(* IEC 61131-3 sources: volt/packages/volt-lsp-iec/test-corpus/lenze-mid/Device/Plc Logic/Application/Library Manager/(unresolved)/iecvaraccessopcuametadata interfaces, 4 files *)

(* ---- VARACCUANAMESPACEFRAGMENT.dut ---- *)
TYPE VARACCUANAMESPACEFRAGMENT :
STRUCT
	FRAGMENTNAMESPACE : POINTER TO OpcUa_String;
	NAMESPACES : POINTER TO OpcUa_String;
	NUMNAMESPACES : UDINT;
	NODES : POINTER TO OpcUaServerNodeDescription;
	NUMNODES : UDINT;
	REFERENCES : POINTER TO OpcUaServerReferenceDescription;
	NUMREFERENCES : UDINT;
	NAMESPACESMAPPED : BOOL;
	INVALIDFRAGMENT : BOOL;
	REFCOUNT : UDINT;
END_STRUCT
END_TYPE

(* ---- INTERFACEIDS.gvl ---- *)
VAR_GLOBAL
	ITFID_IIECVARACCESSOPCUAMETADATA : DWORD := 16#C0;
	ITFID_IIECVARACCESSOPCUAFINDBYBROWSENAME : DWORD := 16#D1;
END_VAR

(* ---- IIECVARACCESSOPCUAFINDBYBROWSENAME.itf ---- *)
INTERFACE IIECVARACCESSOPCUAFINDBYBROWSENAME
END_INTERFACE

METHOD VARACCGETCHILDBYBROWSENAME : IBaseTreeNode
VAR_INPUT
	HNODE : RTS_IEC_HANDLE;
	PVARIABLEINFORMATION : POINTER TO VariableInformationStruct2;
	PBROWSENAME : POINTER TO OpcUa_QualifiedName;
	PRESULT : POINTER TO UDINT;
END_VAR
END_METHOD

METHOD VARACCGETNEXTBYBROWSENAME : IBaseTreeNode
VAR_INPUT
	HNODE : RTS_IEC_HANDLE;
	PVARIABLEINFORMATION : POINTER TO VariableInformationStruct2;
	PBROWSENAME : POINTER TO OpcUa_QualifiedName;
	PRESULT : POINTER TO UDINT;
END_VAR
END_METHOD

(* ---- IIECVARACCESSOPCUAMETADATA.itf ---- *)
INTERFACE IIECVARACCESSOPCUAMETADATA
END_INTERFACE

METHOD VARACCGETUAINFORMATIONMODEL : RTS_IEC_RESULT
VAR_OUTPUT
	NAMESPACES : POINTER TO OpcUa_String;
	NUMNAMESPACES : UDINT;
	FRAGMENTS : POINTER TO POINTER TO VarAccUaNamespaceFragment;
	NUMFRAGMENTS : UDINT;
END_VAR
END_METHOD

METHOD VARACCGETUANAMESPACE : RTS_IEC_RESULT
VAR_OUTPUT
	PMODELNAMESPACE : POINTER TO OpcUa_String;
END_VAR
END_METHOD

METHOD VARACCGETUAENTRYPOINTS : RTS_IEC_RESULT
VAR_OUTPUT
	ENTRYPOINTS : POINTER TO OpcUa_NodeId;
	NUMENTRYPOINTS : UDINT;
END_VAR
END_METHOD

METHOD VARACCGETUAMETHODARGUMENTS : RTS_IEC_RESULT
VAR_INPUT
	HNODE : RTS_IEC_HANDLE;
	PVARINFO : POINTER TO VariableInformationStruct2;
END_VAR
VAR_OUTPUT
	PINPUTARGUMENTS : POINTER TO OpcUa_NodeId;
	POUTPUTARGUMENTS : POINTER TO OpcUa_NodeId;
END_VAR
END_METHOD

METHOD VARACCGETUAENTRYPOINT : RTS_IEC_RESULT
VAR_INPUT
	HNODE : RTS_IEC_HANDLE;
	PVARINFO : POINTER TO VariableInformationStruct2;
END_VAR
VAR_OUTPUT
	ISENTRYPOINT : BOOL;
	PENTRYPOINT : POINTER TO OpcUa_NodeId;
END_VAR
END_METHOD

METHOD VARACCGETUAPARENTREFERENCETYPE : RTS_IEC_RESULT
VAR_INPUT
	HNODE : RTS_IEC_HANDLE;
	PVARINFO : POINTER TO VariableInformationStruct2;
END_VAR
VAR_OUTPUT
	PREFERENCETYPE : POINTER TO OpcUa_NodeId;
END_VAR
END_METHOD

METHOD VARACCGETUATYPEDEFINITION : RTS_IEC_RESULT
VAR_INPUT
	HNODE : RTS_IEC_HANDLE;
	PVARINFO : POINTER TO VariableInformationStruct2;
END_VAR
VAR_OUTPUT
	PTYPEDEFINITION : POINTER TO OpcUa_NodeId;
END_VAR
END_METHOD

METHOD VARACCGETUANODECLASS : RTS_IEC_RESULT
VAR_INPUT
	HNODE : RTS_IEC_HANDLE;
	PVARINFO : POINTER TO VariableInformationStruct2;
END_VAR
VAR_OUTPUT
	NODECLASS : OpcUa_NodeClass;
END_VAR
END_METHOD

METHOD VARACCGETUAEVENTNOTIFIER : RTS_IEC_RESULT
VAR_INPUT
	HNODE : RTS_IEC_HANDLE;
	PVARINFO : POINTER TO VariableInformationStruct2;
END_VAR
VAR_OUTPUT
	EVENTNOTIFIER : OpcUa_Byte;
END_VAR
END_METHOD

METHOD VARACCGETUABROWSENAME : RTS_IEC_RESULT
VAR_INPUT
	HNODE : RTS_IEC_HANDLE;
	PVARINFO : POINTER TO VariableInformationStruct2;
END_VAR
VAR_OUTPUT
	PBROWSENAME : POINTER TO OpcUa_QualifiedName;
END_VAR
END_METHOD

METHOD VARACCGETUADESCRIPTION : RTS_IEC_RESULT
VAR_INPUT
	HNODE : RTS_IEC_HANDLE;
	PVARINFO : POINTER TO VariableInformationStruct2;
END_VAR
VAR_OUTPUT
	PDESCRIPTION : POINTER TO OpcUa_LocalizedText;
END_VAR
END_METHOD

METHOD VARACCGETUADISPLAYNAME : RTS_IEC_RESULT
VAR_INPUT
	HNODE : RTS_IEC_HANDLE;
	PVARINFO : POINTER TO VariableInformationStruct2;
END_VAR
VAR_OUTPUT
	PDISPLAYNAME : POINTER TO OpcUa_LocalizedText;
END_VAR
END_METHOD

METHOD VARACCGETUATYPEDATATYPEID : RTS_IEC_RESULT
VAR_INPUT
	HTYPENODE : RTS_IEC_HANDLE;
END_VAR
VAR_OUTPUT
	PDATATYPEID : POINTER TO OpcUa_NodeId;
END_VAR
END_METHOD

METHOD VARACCGETUATYPEPARENTREFERENCETYPE : RTS_IEC_RESULT
VAR_INPUT
	HTYPENODE : RTS_IEC_HANDLE;
END_VAR
VAR_OUTPUT
	PPARENTREFERENCETYPE : POINTER TO OpcUa_NodeId;
END_VAR
END_METHOD

METHOD VARACCGETUATYPEISWELLKNOWN : RTS_IEC_RESULT
VAR_INPUT
	HTYPENODE : RTS_IEC_HANDLE;
END_VAR
VAR_OUTPUT
	BWELLKNOWN : BOOL;
END_VAR
END_METHOD

METHOD VARACCGETUATYPEPARENTNODE : RTS_IEC_RESULT
VAR_INPUT
	HTYPENODE : RTS_IEC_HANDLE;
END_VAR
VAR_OUTPUT
	PPARENTNODEID : POINTER TO OpcUa_NodeId;
END_VAR
END_METHOD

METHOD VARACCGETUATYPEENCODINGID : RTS_IEC_RESULT
VAR_INPUT
	HTYPENODE : RTS_IEC_HANDLE;
END_VAR
VAR_OUTPUT
	PENCODINGID : POINTER TO OpcUa_NodeId;
END_VAR
END_METHOD
